		E_PMLState.ePMLState_Held:
			Alarms[E_PackMLBase_Alarms.StateHeldEnter].Clear(0, 0);

		E_PMLState.ePMLState_Unholding:
			Alarms[E_PackMLBase_Alarms.StateUnholdingEnter].Clear(0, 0);

		E_PMLState.ePMLState_Suspending:
			Alarms[E_PackMLBase_Alarms.StateSuspendingEnter].Clear(0, 0);

		E_PMLState.ePMLState_Suspended:
			Alarms[E_PackMLBase_Alarms.StateSuspendedEnter].Clear(0, 0);

		E_PMLState.ePMLState_Unsuspending:
			Alarms[E_PackMLBase_Alarms.StateUnsuspendingEnter].Clear(0, 0);

		E_PMLState.ePMLState_Stopping:
			Alarms[E_PackMLBase_Alarms.StateStoppingEnter].Clear(0, 0);

		E_PMLState.ePMLState_Stopped:
			Alarms[E_PackMLBase_Alarms.StateStoppedEnter].Clear(0, 0);

		E_PMLState.ePMLState_Aborting:
			Alarms[E_PackMLBase_Alarms.StateAbortingEnter].Clear(0, 0);

		E_PMLState.ePMLState_Aborted:
			Alarms[E_PackMLBase_Alarms.StateAbortedEnter].Clear(0, 0);

		E_PMLState.ePMLState_Clearing:
			Alarms[E_PackMLBase_Alarms.StateClearingEnter].Clear(0, 0);

		E_PMLState.ePMLState_Undefined:
			Alarms[E_PackMLBase_Alarms.StateUndefinedEnter].Clear(0, 0);
	END_CASE

	LastState := State; //Store previous state
END_IF

(*! <description> The current state is compared against the mode during the last call.  The corresponding events are raised/cleared as the state is changed.
<b>This FB is called from FB_PMLModuleBase.StateControl.  Further calls are not necessary.</b></description>*)

END_FUNCTION_BLOCK

// PackML/FB_PackML_ModeLogger
//! @summary This FB raises events corresponding to <b>mode</b> changes within the parent PackML module
FUNCTION_BLOCK FB_PackML_ModeLogger
VAR_IN_OUT
	Alarms : ARRAY[1..48] OF FB_TcAlarm; //! Array of alarms for Core PackML events that exist in any PackML enabled module
END_VAR

VAR_INPUT
	ModulePrefix : STRING; //! Prefix String for any  <TODO> Remove this? </TODO>
	Mode		 : DINT;   //! Current mode of the module
END_VAR

VAR
	LastMode : DINT;
END_VAR

IF Mode <> LastMode THEN
	CASE Mode OF
		E_PMLUnitMode.ePMLUnitMode_Invalid:
			Alarms[E_PackMLBase_Alarms.ModeInvalidEnter].Raise(0);

		E_PMLUnitMode.ePMLUnitMode_Production:
			Alarms[E_PackMLBase_Alarms.ModeProductionEnter].Raise(0);

		E_PMLUnitMode.ePMLUnitMode_Maintenance:
			Alarms[E_PackMLBase_Alarms.ModeMaintenanceEnter].Raise(0);

		E_PMLUnitMode.ePMLUnitMode_Manual:
			Alarms[E_PackMLBase_Alarms.ModeManualEnter].Raise(0);
	END_CASE

	CASE LastMode OF
		E_PMLUnitMode.ePMLUnitMode_Invalid:
			Alarms[E_PackMLBase_Alarms.ModeInvalidEnter].Clear(0, 0);

		E_PMLUnitMode.ePMLUnitMode_Production:
			Alarms[E_PackMLBase_Alarms.ModeProductionEnter].Clear(0, 0);

		E_PMLUnitMode.ePMLUnitMode_Maintenance:
			Alarms[E_PackMLBase_Alarms.ModeMaintenanceEnter].Clear(0, 0);

		E_PMLUnitMode.ePMLUnitMode_Manual:
			Alarms[E_PackMLBase_Alarms.ModeManualEnter].Clear(0, 0);
	END_CASE

	LastMode := Mode;
END_IF

(*! <description> The current mode is compared against the mode during the last call.  The corresponding events are raised/cleared as the mode is changed.
<b>This FB is called from FB_PMLModuleBase.ModeControl.  Further calls are not necessary.</b></description>*)

END_FUNCTION_BLOCK

// Project Information/F_GetCompany
// This function has been automatically generated from the project information.
{attribute 'signature_flag' := '1073741824'}
{attribute 'TcGenerated'}
{attribute 'no-analysis'}
FUNCTION F_GetCompany : WSTRING
VAR_INPUT
	
END_VAR

F_GetCompany := "Beckhoff Automation LLC";

END_FUNCTION

// Project Information/F_GetTitle
// This function has been automatically generated from the project information.
{attribute 'signature_flag' := '1073741824'}
{attribute 'TcGenerated'}
{attribute 'no-analysis'}
FUNCTION F_GetTitle : WSTRING
VAR_INPUT
	
END_VAR

F_GetTitle := "SPT Base Types";

END_FUNCTION

// Project Information/F_GetVersion
// This function has been automatically generated from the project information.
{attribute 'signature_flag' := '1073741824'}
{attribute 'TcGenerated'}
{attribute 'no-analysis'}
FUNCTION F_GetVersion : ST_LibVersion
VAR_INPUT
	
END_VAR

F_GetVersion.iMajor := 3;
F_GetVersion.iMinor := 2;
F_GetVersion.iBuild := 10;
F_GetVersion.iRevision := 0;
F_GetVersion.sVersion := '3.2.10';
F_GetVersion.nFlags := 1;

END_FUNCTION

// Tracing/FB_TraceLog
FUNCTION_BLOCK FINAL FB_TraceLog
VAR
	Event						 : FB_TcMessage;
	JsonParser					 : FB_JsonDomParser;
	TimeFormatter				 : FB_FormatString;
	MessagesSentThisScan		 : UDINT;
	Previous_AddEntrySource		 : T_MaxString;
	Previous_AddEntryMessage	 : T_MaxString;
	Previous_AddEntryFlags		 : UDINT;
	Previous_AddEntryJsonSource	 : T_MaxString;
	Previous_AddEntryJsonMessage : T_MaxString;
	Previous_AddEntryJsonFlags	 : UDINT;
	Previous_AddEntryJson		 : T_MaxString;
	InitComplete				 : BOOL := FALSE;
END_VAR

METHOD PRIVATE AddContext
VAR_INPUT
	Source : T_MaxString;
	Flags  : UDINT;
END_VAR

VAR
	CurrentDCTime : DCTIMESTRUCT;
	DCTime100Nsec : WORD;
END_VAR
//Collect DC timestamp info and properly format string
CurrentDCTime := DCTIME64_TO_DCTIMESTRUCT(F_GetActualDcTime64());
DCTime100Nsec := CurrentDCTime.wNanoseconds / 100;
TimeFormatter(sFormat := '%2.2d:%2.2d:%2.2d.%3.3d%3.3d%1.1d',
			  arg1	  := F_WORD(CurrentDCTime.wHour),
			  arg2	  := F_WORD(CurrentDCTime.wMinute),
			  arg3	  := F_WORD(CurrentDCTime.wSecond),
			  arg4	  := F_WORD(CurrentDCTime.wMilliseconds),
			  arg5	  := F_WORD(CurrentDCTime.wMicroseconds),
			  arg6	  := F_WORD(DCTime100Nsec));

Event.ipArguments.AddString(TimeFormatter.sOut);												 //DC Timestamp string
Event.ipArguments.AddString(Source);															 //POU calling the Trace() function -- this should come automatically
Event.ipArguments.AddString(TwinCAT_SystemInfoVarList._TaskInfo[GETCURTASKINDEXEX()].TaskName);	 //Task which called the POU last
Event.ipArguments.AddUDInt(TwinCAT_SystemInfoVarList._TaskInfo[GETCURTASKINDEXEX()].CycleCount); //Cycle count of above task
Event.ipArguments.AddUDInt(Flags);																 //General-use flags (application dependent)
END_METHOD

METHOD PUBLIC AddEntry
VAR_INPUT
	Source	: T_MaxString;
	Message : T_MaxString;
	Flags	: UDINT;
END_VAR
IF NOT InitComplete THEN
	RETURN;
END_IF

{analysis -62}
IF NOT TracingAllowed THEN
	{analysis -90}
	RETURN;
END_IF

IF NOT Parameters_Tracing.ALLOW_DUPLICATE_SEQUENTIAL_MESSAGES THEN
	IF (Source = Previous_AddEntrySource) AND (Message = Previous_AddEntryMessage) AND (Flags = Previous_AddEntryFlags) THEN
		//This message is identical to the last message sent--ignore
		RETURN;
	END_IF
END_IF

Event.ipArguments.Clear().AddString(Message);
AddContext(Source := Source, Flags := Flags);
Event.Send(0);
MessagesSentThisScan := MessagesSentThisScan + 1;
MEMSET(ADR(Previous_AddEntrySource), 0, SIZEOF(T_MaxString));
MEMSET(ADR(Previous_AddEntryMessage), 0, SIZEOF(T_MaxString));
Previous_AddEntrySource	 := Source;
Previous_AddEntryMessage := Message;
Previous_AddEntryFlags	 := Flags;
END_METHOD

METHOD PUBLIC AddEntryWithJson
VAR_INPUT
	Source	: T_MaxString;
	Message : T_MaxString;
	Flags	: UDINT;
	Json	: T_MaxString;
END_VAR

VAR
	Document	  : SJsonValue;
	JsonAttribute : T_MaxString;
	TaskName	  : T_MaxString;
	temp		  : udint;
END_VAR

VAR_INST
	LastScanCount		 : UDINT;
	MessagesSentThisScan : UDINT;
	MissedMessages		 : UDINT;
	Throttled			 : BOOL;
END_VAR

VAR
	ThrottledNotificationString : T_MaxString;
	CurrentDCTime				: DCTIMESTRUCT;
	DCTime100Nsec				: WORD;
	DCTimeString				: T_MaxString;
END_VAR
IF NOT InitComplete THEN
	RETURN;
END_IF

{analysis -62}
IF NOT TracingAllowed THEN
	RETURN;
END_IF

IF NOT Parameters_Tracing.ALLOW_DUPLICATE_SEQUENTIAL_MESSAGES THEN
	IF (MEMCMP(ADR(Source), ADR(Previous_AddEntryJsonSource), SIZEOF(T_MaxString)) = 0) AND (MEMCMP(ADR(Message), ADR(Previous_AddEntryJsonMessage), SIZEOF(T_MaxString)) = 0) AND (Flags = Previous_AddEntryJsonFlags) AND (MEMCMP(ADR(Json), ADR(Previous_AddEntryJson), SIZEOF(T_MaxString)) = 0) THEN
		//This message is identical to the last message sent--ignore
		RETURN;
	END_IF
END_IF

Event.ipArguments.Clear().AddString(Message);
AddContext(Source := Source, Flags := Flags);
Document := JsonParser.NewDocument();
JsonParser.AddJsonMember(Document, 'ExtendedInfo', Json);
JsonAttribute := JsonParser.GetJson(Document);
Event.SetJsonAttribute(JsonAttribute);
Event.Send(0);
MessagesSentThisScan := MessagesSentThisScan + 1;
MEMCPY(ADR(Previous_AddEntryJsonSource), ADR(Source), SIZEOF(T_MaxString));
MEMCPY(ADR(Previous_AddEntryJsonMessage), ADR(Message), SIZEOF(T_MaxString));
Previous_AddEntryFlags := Flags;
MEMCPY(ADR(Previous_AddEntryJsonMessage), ADR(Json), SIZEOF(T_MaxString));
END_METHOD

METHOD FB_init : BOOL
VAR_INPUT
	bInitRetains : BOOL; // if TRUE, the retain variables are initialized (warm start / cold start)
	bInCopyCode	 : BOOL; // if TRUE, the instance afterwards gets moved into the copy code (online change)
END_VAR

VAR
	hr : HRESULT;
END_VAR
{analysis -15}
IF NOT Event.EqualsToEventEntryEx(TC_EVENTS.Tracing.TraceEvent) THEN
	IF SUCCEEDED(Event.CreateEx(TC_EVENTS.Tracing.TraceEvent, 0)) THEN
		InitComplete := TRUE;
	END_IF
ELSE
	InitComplete := TRUE;
END_IF
END_METHOD

PROPERTY PRIVATE TracingAllowed : BOOL
GET
VAR_INST
	LastScanCount  : UDINT;
	MissedMessages : UDINT;
	Throttled	   : BOOL;
END_VAR

VAR
	ThrottledNotificationString : T_MaxString;
END_VAR
{analysis -62}
IF NOT Parameters_Tracing.TRACING_ENABLED THEN
	TracingAllowed := FALSE;
	RETURN;
END_IF

IF TwinCAT_SystemInfoVarList._TaskInfo[GETCURTASKINDEXEX()].CycleCount = LastScanCount THEN
	//Trying to send multiple messages in same scan
	IF Throttled THEN
		MissedMessages := MissedMessages + 1;
		RETURN;
	ELSIF MessagesSentThisScan >= Parameters_Tracing.MAX_LOG_ENTRIES_PER_SCAN AND NOT Throttled THEN
		//Need to throttle messsage queue
		Event.ipArguments.Clear().AddString('Too many messages sent in single scan; tracing throttled.');
		Event.Send(0);
		MissedMessages := MissedMessages + 1;
		Throttled	   := TRUE;
		TracingAllowed := FALSE;
		RETURN;
	ELSE
		TracingAllowed := TRUE;
	END_IF
ELSE
	IF Throttled THEN
		ThrottledNotificationString := CONCAT('Missed ', CONCAT(TO_STRING(MissedMessages), ' throttled messages previously.'));
		Event.ipArguments.Clear().AddString(ThrottledNotificationString);
		Event.Send(0);
		MissedMessages := 0;
	END_IF

	LastScanCount		 := TwinCAT_SystemInfoVarList._TaskInfo[GETCURTASKINDEXEX()].CycleCount;
	MessagesSentThisScan := 0;
	Throttled			 := FALSE;
	TracingAllowed		 := TRUE;
END_IF
END_GET
END_PROPERTY

END_FUNCTION_BLOCK

// VISUs/V_MachineModule
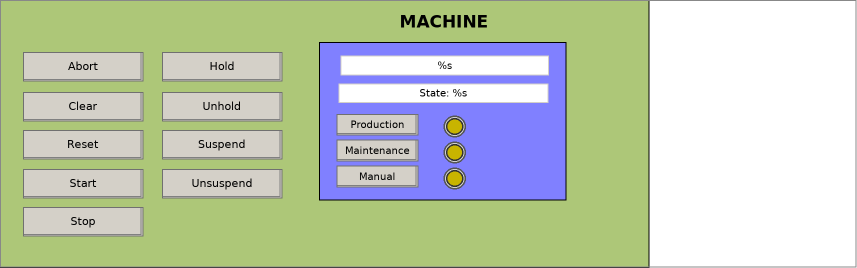
VISUALIZATION V_MachineModule  // 857x268
VAR_IN_OUT
	HMI : ST_PackMLBaseModule_HMI;
END_VAR
    RoundedRectangle (0,0 649x268)
    Button (23,52 120x29), "Abort"
        OnMouseClick: execute { HMI.Command.State := E_PMLCommand.ePMLCommand_Abort; }
    Button (23,92 120x29), "Clear"
        OnMouseClick: execute { HMI.Command.State := E_PMLCommand.ePMLCommand_Clear; }
    Button (23,130 120x29), "Reset"
        OnMouseClick: execute { HMI.Command.State := E_PMLCommand.ePMLCommand_Reset; }
    Button (23,169 120x29), "Start"
        OnMouseClick: execute { HMI.Command.State := E_PMLCommand.ePMLCommand_Start; }
    Button (23,207 120x29), "Stop"
        OnMouseClick: execute { HMI.Command.State := E_PMLCommand.ePMLCommand_Stop; }
    Button (162,52 120x29), "Hold"
        OnMouseClick: execute { HMI.Command.State := E_PMLCommand.ePMLCommand_Hold; }
    Button (162,92 120x29), "Unhold"
        OnMouseClick: execute { HMI.Command.State := E_PMLCommand.ePMLCommand_Unhold; }
    Button (162,130 120x29), "Suspend"
        OnMouseClick: execute { HMI.Command.State := E_PMLCommand.ePMLCommand_Suspend; }
    Button (162,169 120x29), "Unsuspend"
        OnMouseClick: execute { HMI.Command.State := E_PMLCommand.ePMLCommand_Unsuspend; }
    Frame (319,42 247x158)
        shows V_Module(HMI := HMI)
    Label (31,3 826x37), "MACHINE"
END_VISUALIZATION

// VISUs/V_Module
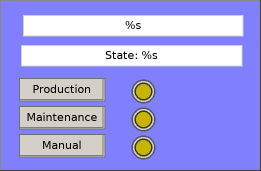
VISUALIZATION V_Module  // 261x171
VAR_IN_OUT
	HMI : ST_PackMLBaseModule_HMI;
END_VAR
    RoundedRectangle (0,0 261x171)
    Textfield (23,15 220x21), "%s", text variable: HMI.Config.Name
    Textfield (21,45 221x21), "State: %s", text variable: HMI.Status.State
    Button (19,78 86x23), "Production"
        OnMouseClick: execute { HMI.Command.Mode := E_PMLUnitMode.ePMLUnitMode_Production; }
    Button (19,106 86x23), "Maintenance"
        OnMouseClick: execute { HMI.Command.Mode := E_PMLUnitMode.ePMLUnitMode_Maintenance; }
    Button (19,134 86x23), "Manual"
        OnMouseClick: execute { HMI.Command.Mode := E_PMLUnitMode.ePMLUnitMode_Manual; }
    Lamp1 (130,78 27x27), variable: HMI.Status.Mode = E_PMLUnitMode.ePMLUnitMode_Production, style: Lamp-Lamp1-Yellow
    Lamp1 (130,106 27x27), variable: HMI.Status.Mode = E_PMLUnitMode.ePMLUnitMode_Maintenance, style: Lamp-Lamp1-Yellow
    Lamp1 (130,134 27x27), variable: HMI.Status.Mode = E_PMLUnitMode.ePMLUnitMode_Manual, style: Lamp-Lamp1-Yellow
END_VISUALIZATION
